(* IEC 61131-3 sources: repolevel_ST_code_completion/dataset/generation_context_ground_truth/ProductionLine, 6 files *)

(* ---- Motor.st ---- *)
VAR
	WaitTimer:TON;
	InternalSequenceDelay:time;
END_VAR

SetFault();
ResetFault();

(* ---- Motor_ResetFault.st ---- *)
VAR
	WaitTimer:TON;
	InternalSequenceDelay:time;
	ResetDetect:r_trig;
END_VAR

ResetDetect(CLK:=MotorI.FaultReset);

IF ResetDetect.Q THEN
	MotorO.FaultStatus:=FALSE;
END_IF

(* ---- Motor_SetFault.st ---- *)
VAR
	WaitTimer:TON;
	InternalSequenceDelay:time;
END_VAR

IF MotorI.Overload THEN
	MotorO.FaultStatus:=TRUE;
	TurnOff();
END_IF

(* ---- Motor_SetWaitTime.st ---- *)
VAR
	WaitTimer:TON;
	InternalSequenceDelay:time;
END_VAR

InternalSequenceDelay:=SequenceDelay;

(* ---- Motor_TurnOff.st ---- *)
VAR
	WaitTimer:TON;
	InternalSequenceDelay:time;
END_VAR

MotorO.Coil:=false;

(* ---- Motor_TurnOn.st ---- *)
VAR
	WaitTimer:TON;
	InternalSequenceDelay:time;
END_VAR

IF MotorO.FaultStatus = FALSE THEN
	WaitTimer(IN:=TRUE , PT:=InternalSequenceDelay);
END_IF

IF WaitTimer.Q THEN
	MotorO.Coil:=TRUE;
	WaitTimer(IN:=FALSE);
END_IF
